// TIA Portal V17 export
// export: Created 2022-06-16T09:21:08.20995Z, ExportSetting WithDefaults, DisplayName Totally Integrated Automation Portal, DisplayVersion V17, DisplayName TIA Portal Openness, DisplayVersion V17, DisplayName TIA Portal Version Control Interface, DisplayVersion V17, DisplayName STEP 7 Professional, DisplayVersion V17, DisplayName STEP 7 Safety, DisplayVersion V17, DisplayName WinCC Advanced, DisplayVersion V17
TYPE "typeAxisParam"
// stored: IsFailsafeCompliant false
   STRUCT
      axisType : String;
      cylinderType : String;
      cylinderDir : Real;
      pistonDiam : Real;
      rodDiam : Real;
      stroke : Real;
      rodPivotPos : Array[1..2] of Real;
      bodyPivotPos : Array[1..2] of Real;
      movingCylinder : Bool;
      angleOffset : Real;
      presDrop : Real;
      nomFlow : Real;
      setpointJump : Real;
      setpointMin : Real;
      sheaveDiam : Real;
      naturalFrequency : Real;
      damping : Real;
   END_STRUCT;
END_TYPE
